(* IEC 61131-3 sources: CodesysTest/export/Testing/HelperFunctions, 7 files *)

(* ---- CheckIfHomed.pou.st ---- *)
(*#-#-#-#-#-#-#-#-#-#---Declaration---#-#-#-#-#-#-#-#-#-#-#-#-#*)

FUNCTION CheckIfHomed : BOOL
VAR_INPUT
	Component : IComponent;
END_VAR
VAR
	homableDevice : IHomable;
END_VAR
(*#-#-#-#-#-#-#-#-#-#---Implementation---#-#-#-#-#-#-#-#-#-#-#-#-#*)

//	Function: CheckIfHomed()
//	Description: Helper function
//				 Pass in a component - if it has a homable motor, and is not yet homed, start homing
//	Created by: Ben Hess
//	Created Date: May 16th, 2019

IF (__QUERYINTERFACE(Component, homableDevice)) THEN
	IF homableDevice.IsHomed OR NOT Component.OptionActive THEN
		CheckIfHomed := TRUE;
	ELSE
		RETURN;
	END_IF
ELSE
	CheckIfHomed := TRUE;
END_IF

(* ---- CheckIfReady.pou.st ---- *)
(*#-#-#-#-#-#-#-#-#-#---Declaration---#-#-#-#-#-#-#-#-#-#-#-#-#*)

FUNCTION CheckIfReady : BOOL
VAR_INPUT
	Component : IComponent;
END_VAR
VAR
END_VAR
(*#-#-#-#-#-#-#-#-#-#---Implementation---#-#-#-#-#-#-#-#-#-#-#-#-#*)

//	Function: CheckIfReady()
//	Description: Helper function
//				 Pass in a component - if it has a homable motor, and is not yet homed, start homing
//	Created by: Ben Hess
//	Created Date: June 13th, 2020

IF Component.Ready OR NOT Component.OptionActive THEN
	CheckIfReady := TRUE;
ELSE
	RETURN;
END_IF

(* ---- ExhaustIfPossible.pou.st ---- *)
(*#-#-#-#-#-#-#-#-#-#---Declaration---#-#-#-#-#-#-#-#-#-#-#-#-#*)

FUNCTION ExhaustIfPossible : BOOL  // Attempts to exhaust SV, returns true if exhaust commanded
VAR_INPUT
	device : IAllObjects;
END_VAR
VAR
	exhaustableDevice : IExhaustable;
END_VAR
(*#-#-#-#-#-#-#-#-#-#---Implementation---#-#-#-#-#-#-#-#-#-#-#-#-#*)

//	Function: ExhaustIfPossible()
//	Description: Helper function
//				 Pass in a device that is controlled byt a SV - exhaust if possible
//	Created by: Ben Hess
//	Created Date: June 25th, 2019

IF (__QUERYINTERFACE(device, exhaustableDevice)) THEN
	exhaustableDevice.Exhaust();
	ExhaustIfPossible := TRUE;
ELSE
	ExhaustIfPossible := FALSE;
END_IF

(* ---- ExtendLPIfPossible.pou.st ---- *)
(*#-#-#-#-#-#-#-#-#-#---Declaration---#-#-#-#-#-#-#-#-#-#-#-#-#*)

FUNCTION ExtendLPIfPossible : BOOL
VAR_INPUT
	device : IAllObjects;
END_VAR
VAR
	extendLowPressureDevice : IExtendLowPressure;
END_VAR
(*#-#-#-#-#-#-#-#-#-#---Implementation---#-#-#-#-#-#-#-#-#-#-#-#-#*)

//	Function: ExtendLPIfPossible()
//	Description: Helper function
//				 Pass in a device that is controlled byt a SV - extend at low pressure if possible
//	Created by: Ben Hess
//	Created Date: June 27th, 2019

IF (__QUERYINTERFACE(device, extendLowPressureDevice)) THEN
	extendLowPressureDevice.ExtendLowPressure();
	ExtendLPIfPossible := TRUE;
ELSE
	ExtendLPIfPossible := FALSE;
END_IF

(* ---- HomeIfNeeded.pou.st ---- *)
(*#-#-#-#-#-#-#-#-#-#---Declaration---#-#-#-#-#-#-#-#-#-#-#-#-#*)

FUNCTION HomeIfNeeded : BOOL
VAR_INPUT
	Component : IComponent;
END_VAR
VAR
	homableDevice : IHomable;
END_VAR
(*#-#-#-#-#-#-#-#-#-#---Implementation---#-#-#-#-#-#-#-#-#-#-#-#-#*)

//	Function: HomeIfNeeded()
//	Description: Helper function
//				 Pass in a component - if it has a homable motor, and is not yet homed, start homing
//	Created by: Ben Hess
//	Created Date: May 16th, 2019

IF (__QUERYINTERFACE(Component, homableDevice)) AND Component.OptionActive THEN
	IF homableDevice.IsHomed THEN
		HomeIfNeeded := TRUE;
		RETURN;
	ELSE
		homableDevice.HomeNow();
	END_IF
END_IF

(* ---- MoveRequested.pou.st ---- *)
(*#-#-#-#-#-#-#-#-#-#---Declaration---#-#-#-#-#-#-#-#-#-#-#-#-#*)

FUNCTION MoveRequested : BOOL
VAR_INPUT
	Component : IComponent;
END_VAR
VAR
	movableDevice : IPostHomeMove;
END_VAR
(*#-#-#-#-#-#-#-#-#-#---Implementation---#-#-#-#-#-#-#-#-#-#-#-#-#*)

//	Function: MoveIfNeeded()
//	Description: Helper function
//				 Pass in a component - if it has a homable motor, and is not yet homed, start homing
//	Created by: Ben Hess
//	Created Date: May 16th, 2019

IF (__QUERYINTERFACE(Component, movableDevice)) AND Component.OptionActive THEN
	IF NOT movableDevice.InDesiredPosition THEN
		MoveRequested := TRUE;
		RETURN;
	ELSE
		RETURN;
	END_IF
END_IF

(* ---- PostHomeMoveIfNeeded.pou.st ---- *)
(*#-#-#-#-#-#-#-#-#-#---Declaration---#-#-#-#-#-#-#-#-#-#-#-#-#*)

FUNCTION PostHomeMoveIfNeeded : BOOL
VAR_INPUT
	Component : IComponent;
END_VAR
VAR
	movableDevice : IPostHomeMove;
END_VAR
(*#-#-#-#-#-#-#-#-#-#---Implementation---#-#-#-#-#-#-#-#-#-#-#-#-#*)

//	Function: MoveIfNeeded()
//	Description: Helper function
//				 Pass in a component - if it has a homable motor, and is homed, and is configured for a post homing move, perform it
//	Created by: Ben Hess
//	Created Date: May 16th, 2019

IF (__QUERYINTERFACE(Component, movableDevice)) AND Component.OptionActive THEN
	IF movableDevice.InDesiredPosition THEN
		PostHomeMoveIfNeeded := TRUE;
		RETURN;
	ELSE
		movableDevice.MoveNow();
	END_IF
END_IF
